TYPE ST_TimedTestState :
STRUCT
    tSafetyTimeout     : TIME;
    nSafetyStartTime   : LWORD;
    bSafetyTimedOut    : BOOL;
    bInitialized       : BOOL;

    nWaitStartTime     : LWORD;
    bWaitComplete      : BOOL;
    bConditionTimedOut : BOOL;
    eWaitType          : E_WaitType;
    tLatchedDuration   : TIME;
END_STRUCT
END_TYPE

(* stored: Version 1.1.0.1
   DUT ST_TimedTestState: Id {9d0fddee-0599-470c-b101-f38bc2c77ade} *)
